INTERFACE ICloneable EXTENDS __System.IQueryInterface

METHOD Clone : IObject
END_METHOD

END_INTERFACE

(* stored: Version 1.1.0.1
   Itf ICloneable: Id {0a9e2f54-7617-4a5d-8fc2-962082da80fb}
   Method Clone: Id {211c847f-0aa0-451e-bc77-9b18b7b131b9} *)
